FUNCTION_BLOCK FB_CoolDownState IMPLEMENTS I_State
VAR_INPUT
END_VAR
VAR_OUTPUT
END_VAR
VAR
	pMachine : POINTER TO FB_StateMachine;	
END_VAR

{warning 'Eigenschaftenimplementierung hinzufügen'}
PROPERTY Description : STRING
GET
Description := 'Heat pump is cooling down';
END_GET
END_PROPERTY

METHOD ErrorDetected : BOOL
VAR_INPUT
	errorEvents		: ST_ErrorEvents;
END_VAR
VAR
	message				: STRING(255);
END_VAR
message := toErrorText(errorEvents);
ADSLOGSTR(ADSLOG_MSGTYPE_HINT, 'Error detected', message);
pMachine^.SetState(pMachine^.ErrorState);
END_METHOD

//FB_Init ist immer implizit verfügbar und wird primär für die Initialisierung verwendet.
//Der Rückgabewert wird nicht ausgewertet. Für gezielte Einflussnahme können Sie
//die Methoden explizit deklarieren und darin mit dem Standard-Initialisierungscode 
//zusätzlichen Code bereitstellen. Sie können den Rückgabewert auswerten.
METHOD FB_Init: BOOL
VAR_INPUT    
	bInitRetains: BOOL; // TRUE: Die Retain-Variablen werden initialisiert (Reset warm / Reset kalt)    
	bInCopyCode: BOOL;  // TRUE: Die Instanz wird danach in den Kopiercode kopiert (Online-Change)
	pMachine : POINTER TO FB_StateMachine;
END_VAR
THIS^.pMachine := pMachine;
END_METHOD

{warning 'Methodenimplementierung hinzufügen'}
METHOD HeatIsRequested : BOOL
END_METHOD

{warning 'Methodenimplementierung hinzufügen'}
METHOD LimitValuesAreExceeded : BOOL
END_METHOD

PROPERTY State : E_State
GET
State := E_State.COOLDOWN;
END_GET
END_PROPERTY

{warning 'Methodenimplementierung hinzufügen'}
METHOD TargetTemeperatureReached : BOOL
END_METHOD

{warning 'Methodenimplementierung hinzufügen'}
METHOD UserPressedConfirmationButton : BOOL
END_METHOD

{warning 'Methodenimplementierung hinzufügen'}
METHOD UserPressedSwitchOffButton : BOOL
END_METHOD

{warning 'Methodenimplementierung hinzufügen'}
METHOD UserPressedSwitchOnButton : BOOL
END_METHOD

{warning 'Methodenimplementierung hinzufügen'}
METHOD WaterHasCooledDown : BOOL
ADSLOGSTR(ADSLOG_MSGTYPE_HINT, 'Abkühlungsphase beendet', pMachine^.iState.Description);
pMachine^.SetState(pMachine^.IdleState);
END_METHOD

END_FUNCTION_BLOCK

(* stored: Version 1.1.0.1
   POU FB_CoolDownState: Id {69543f7c-5310-4c1a-8812-b3e2ffab4bfe}, SpecialFunc None
   Property Description: Id {76a23e04-76c5-464c-a2ea-a1fe64ea1c1f}
   Get Get: Id {48ed62c6-46f8-4900-a687-57fd823269ad}
   Method ErrorDetected: Id {04bb140a-5d6b-4e66-849a-6791cd9086da}
   Method FB_init: Id {63e5eb1b-d453-4548-affe-ff9f484d55b7}
   Method HeatIsRequested: Id {256700ac-59a8-426d-b37d-3bd3eeacc152}
   Method LimitValuesAreExceeded: Id {d817e72e-1f23-4e30-8d38-46e62e4b0873}
   Property State: Id {a82d8201-9208-4f93-83b5-3fa1aefa63ed}
   Get Get: Id {a2871b6a-006c-421a-9886-583166f3d8ff}
   Method TargetTemeperatureReached: Id {660c57e7-0ee7-4900-9c79-b8fdca4c4354}
   Method UserPressedConfirmationButton: Id {a58397d8-89f0-423c-a188-d24ebab8593b}
   Method UserPressedSwitchOffButton: Id {98a471af-99db-479f-bdc4-364d930673d4}
   Method UserPressedSwitchOnButton: Id {8d0ae532-2916-4cc2-8c07-c9276e97bac4}
   Method WaterHasCooledDown: Id {b15859b9-dd1d-425a-9c19-1eb430d81055} *)
